// TIA Portal V17 export
// export: Created 2022-03-30T18:21:29.7902827Z, ExportSetting WithDefaults, DisplayName Totally Integrated Automation Portal, DisplayVersion V17, DisplayName TIA Portal Openness, DisplayVersion V17, DisplayName TIA Portal Version Control Interface, DisplayVersion V17, DisplayName STEP 7 Professional, DisplayVersion V17, DisplayName STEP 7 Safety, DisplayVersion V17, DisplayName WinCC Advanced / Unified PC, DisplayVersion V17
VAR_GLOBAL   // PLC tag table "Default tag table"
   System_Byte AT %MB0 : Byte;
   FirstScan AT %M0.0 : Bool;
   DiagStatusUpdate AT %M0.1 : Bool;
   AlwaysTRUE AT %M0.2 : Bool;
   AlwaysFALSE AT %M0.3 : Bool;
   Clock_Byte AT %MB1 : Byte;
   Clock_10Hz AT %M1.0 : Bool;
   Clock_5Hz AT %M1.1 : Bool;
   "Clock_2.5Hz" AT %M1.2 : Bool;
   Clock_2Hz AT %M1.3 : Bool;
   "Clock_1.25Hz" AT %M1.4 : Bool;
   Clock_1Hz AT %M1.5 : Bool;
   "Clock_0.625Hz" AT %M1.6 : Bool;
   "Clock_0.5Hz" AT %M1.7 : Bool;
   bx_EM00_CM02_PalletSensor AT %I0.0 : Bool;
   by_EM00_CM02_ConvFrd AT %Q0.0 : Bool;
   bx_EM00_CM03_PalletSensor AT %I0.1 : Bool;
   by_EM00_CM03_RollsFrd AT %Q0.1 : Bool;
   by_EM00_CM03_RollsRev AT %Q0.2 : Bool;
   by_EM00_CM03_ChainFrd AT %Q0.3 : Bool;
   by_EM00_CM03_ChainRev AT %Q0.4 : Bool;
   by_EM00_CM04_ConvFrd AT %Q0.5 : Bool;
   bx_EM01_CM01_BoxSensor AT %I0.3 : Bool;
   by_EM01_CM01_BeltFrd AT %Q0.6 : Bool;
   Tag_12 AT %I0.4 : Bool;
   bx_EM01_CM02_PalletSensor1 AT %I0.5 : Bool;
   bx_EM01_CM02_PalletSensor2 AT %I0.6 : Bool;
   bx_EM01_CM02_PusherInPos AT %I0.7 : Bool;
   bx_EM01_CM02_TrapdoorInPos AT %I1.0 : Bool;
   bx_EM01_CM02_PositionerExtended AT %I1.1 : Bool;
   bx_EM01_CM02_LiftMoving AT %I1.2 : Bool;
   by_EM01_CM02_BeltFrd AT %Q0.7 : Bool;
   by_EM01_CM02_BeltRev AT %Q1.0 : Bool;
   by_EM01_CM02_Pusher AT %Q1.1 : Bool;
   by_EM01_CM02_Positioner AT %Q1.2 : Bool;
   by_EM01_CM02_Trapdoor AT %Q1.3 : Bool;
   by_EM01_CM02_MoveLiftToLimit AT %Q1.4 : Bool;
   by_EM01_CM02_LiftUp AT %Q1.5 : Bool;
   by_EM01_CM02_LiftDown AT %Q1.6 : Bool;
   by_EM01_CM02_ChainFrd AT %Q1.7 : Bool;
   by_EM01_CM02_ChainRev AT %Q2.0 : Bool;
   by_EM00_CM03_ChainRollsFrd AT %Q2.1 : Bool;
   by_EM00_CM03_ChainRollsRev AT %Q2.2 : Bool;
   by_EM01_CM02_BoxCam AT %Q2.3 : Bool;
   bx_EM00_CM04_PalletSensor AT %I2.2 : Bool;
   by_EM00_CM04_RollsRollsFrd AT %Q4.6 : Bool;
   by_EM00_CM04_RollsRev AT %Q4.7 : Bool;
   by_EM00_CM04_RollsFrd AT %Q5.0 : Bool;
   by_EM00_CM04_ChainFrd AT %Q5.1 : Bool;
   by_EM00_CM04_ChainRev AT %Q5.2 : Bool;
   by_EM00_CM04_ChainRollsFrd AT %Q5.3 : Bool;
   by_EM00_CM04_ChainRollsRev AT %Q5.4 : Bool;
   by_EM00_CM05_RollsFrd AT %Q5.5 : Bool;
   bx_EM02_CM01_BoxSensor AT %I1.5 : Bool;
   by_EM02_CM01_BeltFrd AT %Q3.3 : Bool;
   bx_EM02_CM02_PalletSensor1 AT %I1.7 : Bool;
   bx_EM02_CM02_PalletSensor2 AT %I1.6 : Bool;
   bx_EM02_CM02_PusherInPos AT %I1.4 : Bool;
   bx_EM02_CM02_TrapdoorInPos AT %I2.0 : Bool;
   bx_EM02_CM02_PositionerExtended AT %I2.1 : Bool;
   bx_EM02_CM02_LiftMoving AT %I1.3 : Bool;
   by_EM02_CM02_BeltFrd AT %Q3.4 : Bool;
   by_EM02_CM02_BeltRev AT %Q99.0 : Bool;
   by_EM02_CM02_Pusher AT %Q3.6 : Bool;
   by_EM02_CM02_Trapdoor AT %Q4.0 : Bool;
   by_EM02_CM02_MoveLiftToLimit AT %Q4.3 : Bool;
   by_EM02_CM02_LiftUp AT %Q4.1 : Bool;
   by_EM02_CM02_LiftDown AT %Q4.2 : Bool;
   by_EM02_CM02_ChainFrd AT %Q4.4 : Bool;
   by_EM02_CM02_ChainRev AT %Q4.5 : Bool;
   by_EM02_CM02_BoxCam AT %Q3.5 : Bool;
   by_EM02_CM02_Positioner AT %Q3.7 : Bool;
END_VAR
